TYPE iol_slave_mlg2prime_output_status_1 :
STRUCT
	q1:							BIT;
	q2:							BIT;
	q3:							BIT;
	q4:							BIT;	
END_STRUCT
END_TYPE

(* stored: Version 1.1.0.1, ProductVersion 3.1.4024.3
   DUT iol_slave_mlg2prime_output_status_1: Id {4f1c9b16-8f93-0feb-3906-8df7ab6b38f1} *)
